FUNCTION F_MultiZError_TO_ErrorId : ERRORID
VAR_INPUT
	nErrorCode	: USINT;
END_VAR
VAR
END_VAR

F_MultiZError_TO_ErrorId := nErrorCode + 41727;

END_FUNCTION

(* stored: Version 1.1.0.1, ProductVersion 3.1.0.25
   POU F_MultiZError_TO_ErrorId: Id {b22e8449-3f00-4007-848b-d7c4a4fd90cb} *)
